(* IEC 61131-3 sources: repolevel_ST_code_completion/output/full_case_fixed/repoeval_Wrappers/readful_result_history, 4 files *)

(* ---- FB_Wrapper_0.st ---- *)
FUNCTION_BLOCK FB_Wrapper
VAR_INPUT
	in:BOOL;
END_VAR
VAR_OUTPUT
	out:BOOL;
END_VAR
VAR
	fb_teste: ARRAY [1..3] OF FB_Teste;
	index: INT;
END_VAR

fb_teste[1].SetTempo(delay := T#4S);
fb_teste[2].SetTempo(delay := T#1S);
fb_teste[3].SetTempo(delay := T#2S);

FOR index := 1 TO 3 DO
	IF in THEN
		fb_teste[index].mLiga();
	ELSE
		fb_teste[index].mDesliga();
	END_IF;
END_FOR;

out := FALSE;
FOR index := 1 TO 3 DO
	IF fb_teste[index].saida THEN
		out := TRUE;
		EXIT;
	END_IF;
END_FOR;
END_FUNCTION_BLOCK

(* ---- FB_Wrapper_1.st ---- *)
FUNCTION_BLOCK FB_Wrapper
VAR_INPUT
	in:BOOL;
END_VAR
VAR_OUTPUT
	out:BOOL;
END_VAR
VAR
	fb_teste: ARRAY [1..3] OF FB_Teste;
	index: INT;
END_VAR

fb_teste[1](delay := T#4S);
fb_teste[2](delay := T#1S);
fb_teste[3](delay := T#2S);

FOR index := 1 TO 3 DO
	IF in THEN
		fb_teste[index].mLiga();
	ELSE
		fb_teste[index].mDesliga();
	END_IF;
END_FOR;

out := FALSE;
FOR index := 1 TO 3 DO
	IF fb_teste[index].saida THEN
		out := TRUE;
		EXIT;
	END_IF;
END_FOR;
END_FUNCTION_BLOCK

(* ---- FB_Wrapper_2.st ---- *)
FUNCTION_BLOCK FB_Wrapper
VAR_INPUT
	in:BOOL;
END_VAR
VAR_OUTPUT
	out:BOOL;
END_VAR
VAR
	fb_teste: ARRAY [1..3] OF FB_Teste;
	index: INT;
END_VAR

fb_teste[1].SetTempo(delay := T#4S);
fb_teste[2].SetTempo(delay := T#1S);
fb_teste[3].SetTempo(delay := T#2S);

FOR index := 1 TO 3 DO
	IF in THEN
		fb_teste[index].mLiga();
	ELSE
		fb_teste[index].mDesliga();
	END_IF;
END_FOR;

out := FALSE;
FOR index := 1 TO 3 DO
	IF fb_teste[index].saida THEN
		out := TRUE;
		EXIT;
	END_IF;
END_FOR;
END_FUNCTION_BLOCK

(* ---- FB_Wrapper_3.st ---- *)
FUNCTION_BLOCK FB_Wrapper
VAR_INPUT
	in:BOOL;
END_VAR
VAR_OUTPUT
	out:BOOL;
END_VAR
VAR
	fb_teste: ARRAY [1..3] OF FB_Teste;
	index: INT;
END_VAR

FOR index := 1 TO 3 DO
  // Set individual delay times based on the index for each FB_Teste instance
  CASE index OF
    1: fb_teste[index].SetTempo(delay := T#4S);
    2: fb_teste[index].SetTempo(delay := T#1S);
    3: fb_teste[index].SetTempo(delay := T#2S);
  END_CASE;

  // Check the input and activate or deactivate the function block
  IF in THEN
    fb_teste[index].mLiga();
  ELSE
    fb_teste[index].mDesliga();
  END_IF;
END_FOR;

out := FALSE;
FOR index := 1 TO 3 DO
  // Check the output of each FB_Teste instance
  IF fb_teste[index].saida THEN
    out := TRUE;
    EXIT;
  END_IF;
END_FOR;
END_FUNCTION_BLOCK
